FUNCTION_BLOCK MultiStation EXTENDS Objective;
VAR_INPUT
	PositionTrigger		: PositionTrigger;
	Station				: ARRAY[0..GVL.MULTISTN_NUM_STN - 1] OF Station;
END_VAR
VAR_OUTPUT
END_VAR
VAR
	i: INT;

    {attribute 'hide'}
    internalPosition : LREAL;
	internalTrackId : DINT; 
END_VAR

{attribute 'monitoring' := 'variable'}
PROPERTY AllMoversInPosition : BOOL
GET
VAR

    i          : ULINT;
	TrackedMovers	: UINT;
END_VAR
// default to false
AllMoversInPosition := TRUE;
TrackedMovers		:= 0;

FOR i := 0 TO SIZEOF(Station) / SIZEOF(Station[0]) - 1 DO
	IF Station[i].TrackedMoverCount > 0 THEN
		TrackedMovers	:= TrackedMovers + 1;
		IF NOT Station[i].MoverInPosition THEN
			AllMoversInPosition	:= FALSE;
			EXIT;
		END_IF
	END_IF
END_FOR

IF TrackedMovers = 0 THEN
	AllMoversInPosition	:= FALSE;
END_IF
END_GET
END_PROPERTY

METHOD Cyclic : BOOL
VAR
	i : USINT;
END_VAR
//IF PositionTrigger.MoverPassedPosition THEN
//	PositionTrigger.CurrentMover.MoveToStation(Station[0]);
//	PositionTrigger.MuteCurrent();
//END_IF

// Call Cyclics
PositionTrigger.Cyclic();
FOR i := 0 TO GVL.MULTISTN_NUM_STN - 1 DO
	Station[i].Cyclic();
END_FOR
END_METHOD

{attribute 'monitoring' := 'call'}
PROPERTY Position : LREAL
GET
InternalPosition	:= Station[0].Position;
Position 			:= internalPosition;
Position;
END_GET
END_PROPERTY

METHOD RegisterMover : BOOL
VAR_INPUT
    NewMover : REFERENCE TO Mover;
END_VAR
(*
	Add a mover to a list of movers tracked by the objective.
	Movers can't be added multiple times, so check for duplicates
	Movers can't overwrite others in the list, so check that the array element is clear
*)
PositionTrigger.RegisterMover(NewMover);
END_METHOD

METHOD RegisterMoverList : BOOL
VAR_INPUT
    NewMoverList : iMoverList;
END_VAR
(*
	Adds an entire MoverList to the Tracked Movers of the objective.
*)

PositionTrigger.RegisterMoverList(NewMoverList);
END_METHOD

PROPERTY TrackId : DINT
GET
TrackId := internalTrackId;
END_GET
SET
internalTrackId := TrackId;
END_SET
END_PROPERTY

METHOD UnregisterAll : BOOL
// Blow out the tracked mover array
PositionTrigger.UnregisterAll();
FOR i := 0 TO GVL.MULTISTN_NUM_STN - 1 DO
	Station[i].UnregisterAll();
END_FOR
END_METHOD

METHOD UnregisterCurrent : BOOL
VAR_INPUT
END_VAR
PositionTrigger.UnregisterCurrent();
END_METHOD

METHOD UnregisterMover : BOOL
VAR_INPUT
    RemovingMover : REFERENCE TO Mover;
END_VAR
PositionTrigger.UnregisterMover(RemovingMover);
END_METHOD

END_FUNCTION_BLOCK

(* stored: Version 1.1.0.1, ProductVersion 3.1.4024.12
   POU MultiStation: Id {df655378-d65d-08eb-0626-40053447c2ec}, SpecialFunc None
   Folder Methods: Id {26448ae6-7421-0b31-2949-700660ed0451}
   Folder Properties: Id {830dba99-a22e-029a-3290-dc45b9f77c2c}
   Property AllMoversInPosition: Id {1f754e83-88fa-0a8d-24cd-753cdf0d29cd}
   Get Get: Id {453286f5-9524-07a2-3f4f-b23cf223a48a}
   Method Cyclic: Id {e1b380b8-f648-0a8a-3ba6-02e42127a4fc}
   Property Position: Id {0439a2f6-0763-0006-1e13-61f08c347974}
   Get Get: Id {8df76152-beee-0302-1b00-ad31e63cb392}
   Method RegisterMover: Id {cd7c1bfa-18cf-06aa-2fce-f8051f74fbc1}
   Method RegisterMoverList: Id {110fc79e-5b4c-0d96-0e95-fb8a117fe6fb}
   Property TrackId: Id {ca736e0d-be92-0876-1f98-2eb101c0025c}
   Get Get: Id {6fa25f0d-0025-0852-0183-6627e2101c7c}
   Set Set: Id {a8dabba8-b7e5-05b5-2515-5c15daaf2851}
   Method UnregisterAll: Id {6fdb2734-0f5a-0fe7-3007-5ae910c9a792}
   Method UnregisterCurrent: Id {464efb4f-da02-0ff6-296e-d86da6fd448b}
   Method UnregisterMover: Id {6f37bac7-c3f6-0993-0d64-9d4d34b88d8b} *)
